// TIA Portal V19 export
FUNCTION "INTERLOCK DB" : Void   // FC17, LAD
{ S7_Optimized_Access := 'TRUE' }
// stored: SetENOAutomatically false
BEGIN

REGION Network 1: ERROR
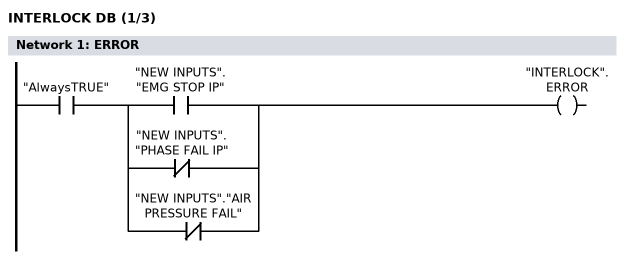
   RUNG wire#powerrail
      Contact( "AlwaysTRUE" )
      wire#w1
      Contact( "NEW INPUTS"."EMG STOP IP" )
      wire#w2
      Coil( "INTERLOCK".ERROR )
   END_RUNG
   RUNG wire#w1
      I_Contact( "NEW INPUTS"."PHASE FAIL IP" )
   END_RUNG wire#w2
   RUNG wire#w1
      I_Contact( "NEW INPUTS"."AIR PRESSURE FAIL" )
   END_RUNG wire#w2
   // the same network as SCL:
   "INTERLOCK".ERROR := "AlwaysTRUE" AND ("NEW INPUTS"."EMG STOP IP" OR NOT "NEW INPUTS"."PHASE FAIL IP" OR NOT "NEW INPUTS"."AIR PRESSURE FAIL");
END_REGION

REGION Network 2: MANUAL RESET
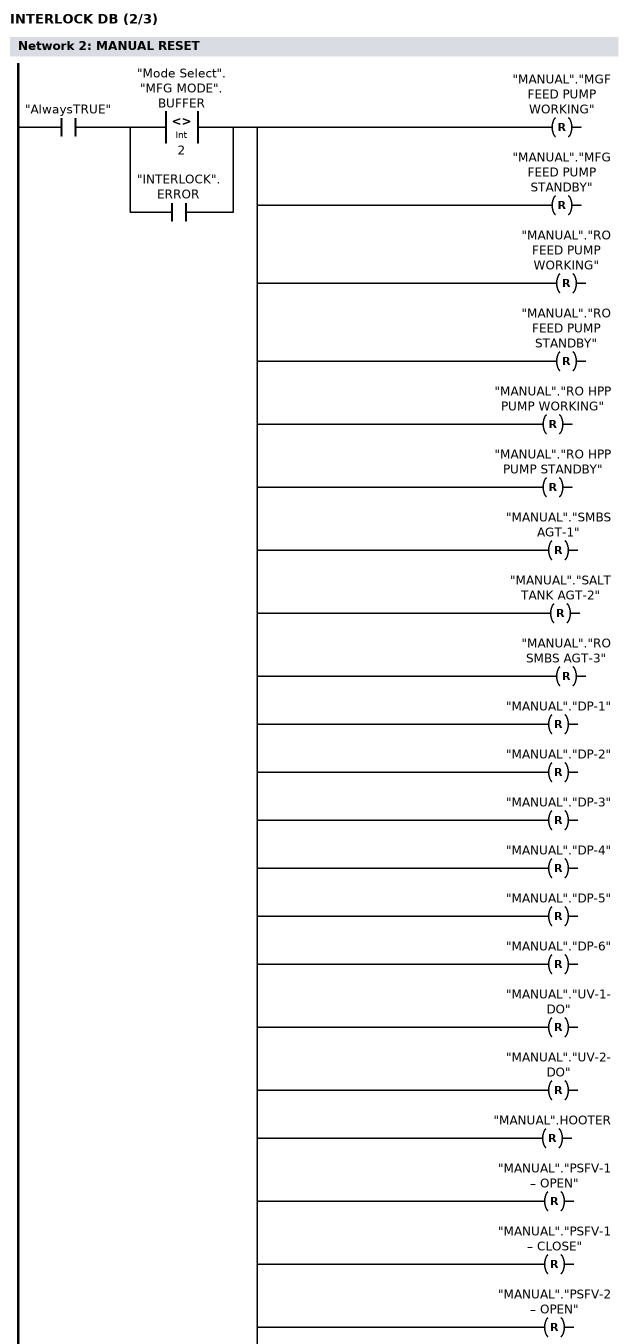
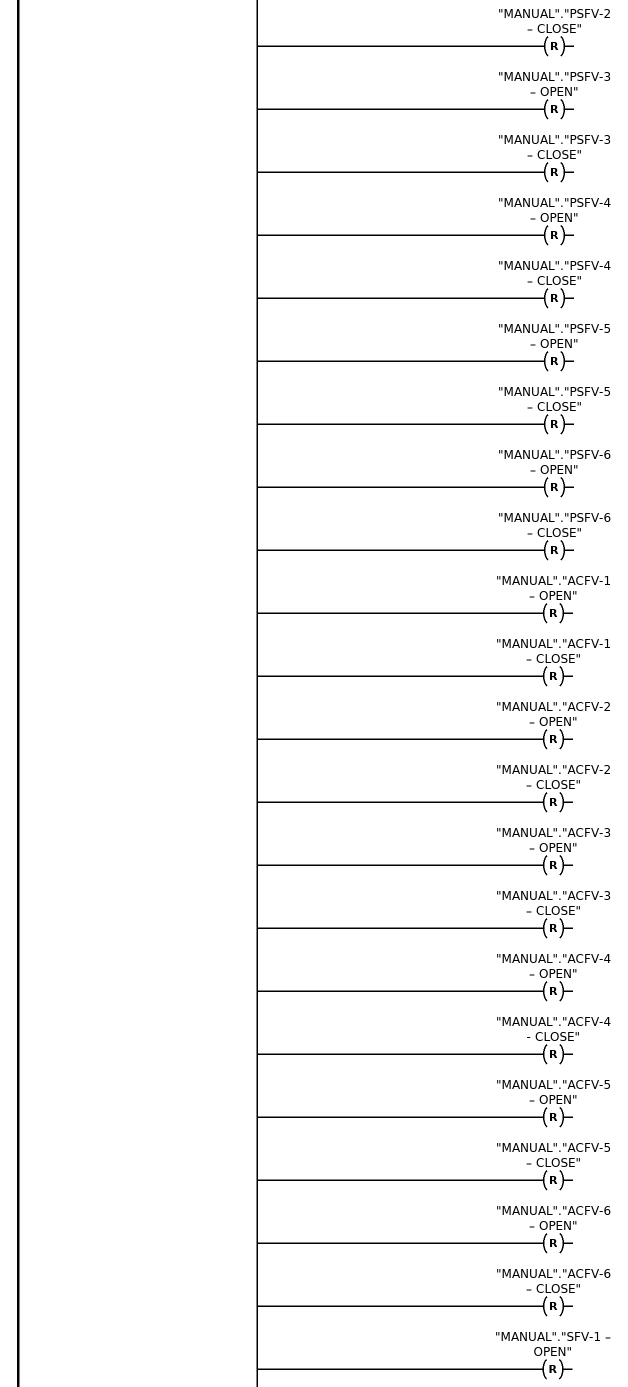
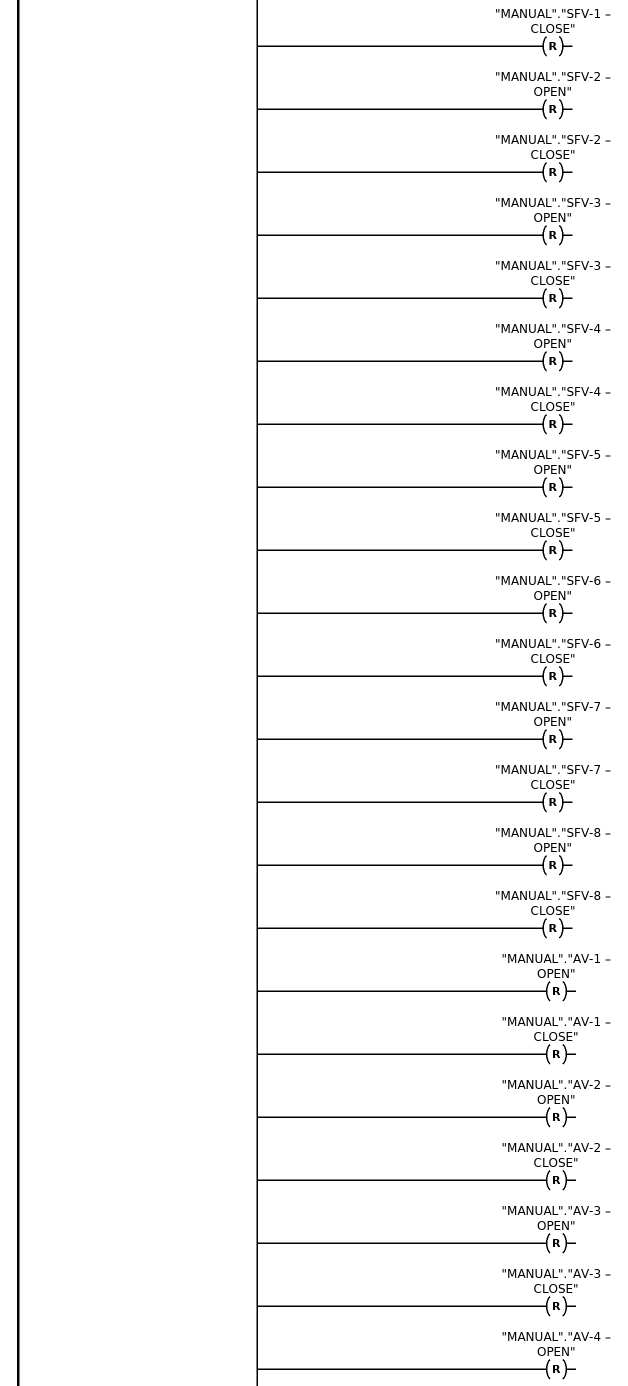
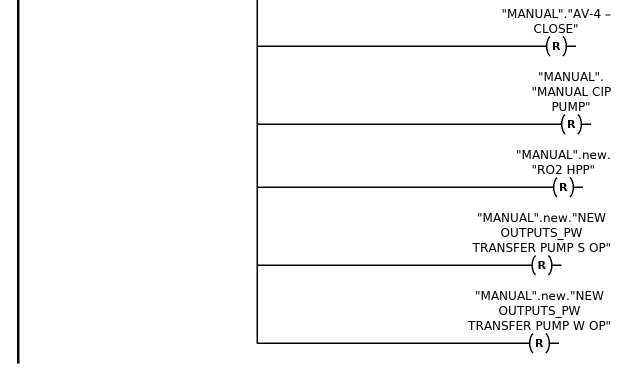
   RUNG wire#powerrail
      Contact( "AlwaysTRUE" )
      wire#w1
      { S7_Templates := "SrcType := Int" } NE_Contact(in1 := "Mode Select"."MFG MODE".BUFFER, in2 := 2)
      wire#w2
      R_Coil( "MANUAL"."MGF FEED PUMP WORKING" )
   END_RUNG
   RUNG wire#w1
      Contact( "INTERLOCK".ERROR )
   END_RUNG wire#w2
   RUNG wire#w2
      R_Coil( "MANUAL"."MFG FEED PUMP STANDBY" )
   END_RUNG
   RUNG wire#w2
      R_Coil( "MANUAL"."RO FEED PUMP WORKING" )
   END_RUNG
   RUNG wire#w2
      R_Coil( "MANUAL"."RO FEED PUMP STANDBY" )
   END_RUNG
   RUNG wire#w2
      R_Coil( "MANUAL"."RO HPP PUMP WORKING" )
   END_RUNG
   RUNG wire#w2
      R_Coil( "MANUAL"."RO HPP PUMP STANDBY" )
   END_RUNG
   RUNG wire#w2
      R_Coil( "MANUAL"."SMBS AGT-1" )
   END_RUNG
   RUNG wire#w2
      R_Coil( "MANUAL"."SALT TANK AGT-2" )
   END_RUNG
   RUNG wire#w2
      R_Coil( "MANUAL"."RO SMBS AGT-3" )
   END_RUNG
   RUNG wire#w2
      R_Coil( "MANUAL"."DP-1" )
   END_RUNG
   RUNG wire#w2
      R_Coil( "MANUAL"."DP-2" )
   END_RUNG
   RUNG wire#w2
      R_Coil( "MANUAL"."DP-3" )
   END_RUNG
   RUNG wire#w2
      R_Coil( "MANUAL"."DP-4" )
   END_RUNG
   RUNG wire#w2
      R_Coil( "MANUAL"."DP-5" )
   END_RUNG
   RUNG wire#w2
      R_Coil( "MANUAL"."DP-6" )
   END_RUNG
   RUNG wire#w2
      R_Coil( "MANUAL"."UV-1-DO" )
   END_RUNG
   RUNG wire#w2
      R_Coil( "MANUAL"."UV-2-DO" )
   END_RUNG
   RUNG wire#w2
      R_Coil( "MANUAL".HOOTER )
   END_RUNG
   RUNG wire#w2
      R_Coil( "MANUAL"."PSFV-1 – OPEN" )
   END_RUNG
   RUNG wire#w2
      R_Coil( "MANUAL"."PSFV-1 – CLOSE" )
   END_RUNG
   RUNG wire#w2
      R_Coil( "MANUAL"."PSFV-2 – OPEN" )
   END_RUNG
   RUNG wire#w2
      R_Coil( "MANUAL"."PSFV-2 – CLOSE" )
   END_RUNG
   RUNG wire#w2
      R_Coil( "MANUAL"."PSFV-3 – OPEN" )
   END_RUNG
   RUNG wire#w2
      R_Coil( "MANUAL"."PSFV-3 – CLOSE" )
   END_RUNG
   RUNG wire#w2
      R_Coil( "MANUAL"."PSFV-4 – OPEN" )
   END_RUNG
   RUNG wire#w2
      R_Coil( "MANUAL"."PSFV-4 – CLOSE" )
   END_RUNG
   RUNG wire#w2
      R_Coil( "MANUAL"."PSFV-5 – OPEN" )
   END_RUNG
   RUNG wire#w2
      R_Coil( "MANUAL"."PSFV-5 – CLOSE" )
   END_RUNG
   RUNG wire#w2
      R_Coil( "MANUAL"."PSFV-6 – OPEN" )
   END_RUNG
   RUNG wire#w2
      R_Coil( "MANUAL"."PSFV-6 – CLOSE" )
   END_RUNG
   RUNG wire#w2
      R_Coil( "MANUAL"."ACFV-1 – OPEN" )
   END_RUNG
   RUNG wire#w2
      R_Coil( "MANUAL"."ACFV-1 – CLOSE" )
   END_RUNG
   RUNG wire#w2
      R_Coil( "MANUAL"."ACFV-2 – OPEN" )
   END_RUNG
   RUNG wire#w2
      R_Coil( "MANUAL"."ACFV-2 – CLOSE" )
   END_RUNG
   RUNG wire#w2
      R_Coil( "MANUAL"."ACFV-3 – OPEN" )
   END_RUNG
   RUNG wire#w2
      R_Coil( "MANUAL"."ACFV-3 – CLOSE" )
   END_RUNG
   RUNG wire#w2
      R_Coil( "MANUAL"."ACFV-4 – OPEN" )
   END_RUNG
   RUNG wire#w2
      R_Coil( "MANUAL"."ACFV-4 - CLOSE" )
   END_RUNG
   RUNG wire#w2
      R_Coil( "MANUAL"."ACFV-5 – OPEN" )
   END_RUNG
   RUNG wire#w2
      R_Coil( "MANUAL"."ACFV-5 – CLOSE" )
   END_RUNG
   RUNG wire#w2
      R_Coil( "MANUAL"."ACFV-6 – OPEN" )
   END_RUNG
   RUNG wire#w2
      R_Coil( "MANUAL"."ACFV-6 – CLOSE" )
   END_RUNG
   RUNG wire#w2
      R_Coil( "MANUAL"."SFV-1 – OPEN" )
   END_RUNG
   RUNG wire#w2
      R_Coil( "MANUAL"."SFV-1 – CLOSE" )
   END_RUNG
   RUNG wire#w2
      R_Coil( "MANUAL"."SFV-2 – OPEN" )
   END_RUNG
   RUNG wire#w2
      R_Coil( "MANUAL"."SFV-2 – CLOSE" )
   END_RUNG
   RUNG wire#w2
      R_Coil( "MANUAL"."SFV-3 – OPEN" )
   END_RUNG
   RUNG wire#w2
      R_Coil( "MANUAL"."SFV-3 – CLOSE" )
   END_RUNG
   RUNG wire#w2
      R_Coil( "MANUAL"."SFV-4 – OPEN" )
   END_RUNG
   RUNG wire#w2
      R_Coil( "MANUAL"."SFV-4 – CLOSE" )
   END_RUNG
   RUNG wire#w2
      R_Coil( "MANUAL"."SFV-5 – OPEN" )
   END_RUNG
   RUNG wire#w2
      R_Coil( "MANUAL"."SFV-5 – CLOSE" )
   END_RUNG
   RUNG wire#w2
      R_Coil( "MANUAL"."SFV-6 – OPEN" )
   END_RUNG
   RUNG wire#w2
      R_Coil( "MANUAL"."SFV-6 – CLOSE" )
   END_RUNG
   RUNG wire#w2
      R_Coil( "MANUAL"."SFV-7 – OPEN" )
   END_RUNG
   RUNG wire#w2
      R_Coil( "MANUAL"."SFV-7 – CLOSE" )
   END_RUNG
   RUNG wire#w2
      R_Coil( "MANUAL"."SFV-8 – OPEN" )
   END_RUNG
   RUNG wire#w2
      R_Coil( "MANUAL"."SFV-8 – CLOSE" )
   END_RUNG
   RUNG wire#w2
      R_Coil( "MANUAL"."AV-1 – OPEN" )
   END_RUNG
   RUNG wire#w2
      R_Coil( "MANUAL"."AV-1 – CLOSE" )
   END_RUNG
   RUNG wire#w2
      R_Coil( "MANUAL"."AV-2 – OPEN" )
   END_RUNG
   RUNG wire#w2
      R_Coil( "MANUAL"."AV-2 – CLOSE" )
   END_RUNG
   RUNG wire#w2
      R_Coil( "MANUAL"."AV-3 – OPEN" )
   END_RUNG
   RUNG wire#w2
      R_Coil( "MANUAL"."AV-3 – CLOSE" )
   END_RUNG
   RUNG wire#w2
      R_Coil( "MANUAL"."AV-4 – OPEN" )
   END_RUNG
   RUNG wire#w2
      R_Coil( "MANUAL"."AV-4 – CLOSE" )
   END_RUNG
   RUNG wire#w2
      R_Coil( "MANUAL"."MANUAL CIP PUMP" )
   END_RUNG
   RUNG wire#w2
      R_Coil( "MANUAL".new."RO2 HPP" )
   END_RUNG
   RUNG wire#w2
      R_Coil( "MANUAL".new."NEW OUTPUTS_PW TRANSFER PUMP S OP" )
   END_RUNG
   RUNG wire#w2
      R_Coil( "MANUAL".new."NEW OUTPUTS_PW TRANSFER PUMP W OP" )
   END_RUNG
   // the same network as SCL:
   IF "AlwaysTRUE" AND (("Mode Select"."MFG MODE".BUFFER <> 2) OR "INTERLOCK".ERROR) THEN
       "MANUAL"."MGF FEED PUMP WORKING" := FALSE;
       "MANUAL"."MFG FEED PUMP STANDBY" := FALSE;
       "MANUAL"."RO FEED PUMP WORKING" := FALSE;
       "MANUAL"."RO FEED PUMP STANDBY" := FALSE;
       "MANUAL"."RO HPP PUMP WORKING" := FALSE;
       "MANUAL"."RO HPP PUMP STANDBY" := FALSE;
       "MANUAL"."SMBS AGT-1" := FALSE;
       "MANUAL"."SALT TANK AGT-2" := FALSE;
       "MANUAL"."RO SMBS AGT-3" := FALSE;
       "MANUAL"."DP-1" := FALSE;
       "MANUAL"."DP-2" := FALSE;
       "MANUAL"."DP-3" := FALSE;
       "MANUAL"."DP-4" := FALSE;
       "MANUAL"."DP-5" := FALSE;
       "MANUAL"."DP-6" := FALSE;
       "MANUAL"."UV-1-DO" := FALSE;
       "MANUAL"."UV-2-DO" := FALSE;
       "MANUAL".HOOTER := FALSE;
       "MANUAL"."PSFV-1 – OPEN" := FALSE;
       "MANUAL"."PSFV-1 – CLOSE" := FALSE;
       "MANUAL"."PSFV-2 – OPEN" := FALSE;
       "MANUAL"."PSFV-2 – CLOSE" := FALSE;
       "MANUAL"."PSFV-3 – OPEN" := FALSE;
       "MANUAL"."PSFV-3 – CLOSE" := FALSE;
       "MANUAL"."PSFV-4 – OPEN" := FALSE;
       "MANUAL"."PSFV-4 – CLOSE" := FALSE;
       "MANUAL"."PSFV-5 – OPEN" := FALSE;
       "MANUAL"."PSFV-5 – CLOSE" := FALSE;
       "MANUAL"."PSFV-6 – OPEN" := FALSE;
       "MANUAL"."PSFV-6 – CLOSE" := FALSE;
       "MANUAL"."ACFV-1 – OPEN" := FALSE;
       "MANUAL"."ACFV-1 – CLOSE" := FALSE;
       "MANUAL"."ACFV-2 – OPEN" := FALSE;
       "MANUAL"."ACFV-2 – CLOSE" := FALSE;
       "MANUAL"."ACFV-3 – OPEN" := FALSE;
       "MANUAL"."ACFV-3 – CLOSE" := FALSE;
       "MANUAL"."ACFV-4 – OPEN" := FALSE;
       "MANUAL"."ACFV-4 - CLOSE" := FALSE;
       "MANUAL"."ACFV-5 – OPEN" := FALSE;
       "MANUAL"."ACFV-5 – CLOSE" := FALSE;
       "MANUAL"."ACFV-6 – OPEN" := FALSE;
       "MANUAL"."ACFV-6 – CLOSE" := FALSE;
       "MANUAL"."SFV-1 – OPEN" := FALSE;
       "MANUAL"."SFV-1 – CLOSE" := FALSE;
       "MANUAL"."SFV-2 – OPEN" := FALSE;
       "MANUAL"."SFV-2 – CLOSE" := FALSE;
       "MANUAL"."SFV-3 – OPEN" := FALSE;
       "MANUAL"."SFV-3 – CLOSE" := FALSE;
       "MANUAL"."SFV-4 – OPEN" := FALSE;
       "MANUAL"."SFV-4 – CLOSE" := FALSE;
       "MANUAL"."SFV-5 – OPEN" := FALSE;
       "MANUAL"."SFV-5 – CLOSE" := FALSE;
       "MANUAL"."SFV-6 – OPEN" := FALSE;
       "MANUAL"."SFV-6 – CLOSE" := FALSE;
       "MANUAL"."SFV-7 – OPEN" := FALSE;
       "MANUAL"."SFV-7 – CLOSE" := FALSE;
       "MANUAL"."SFV-8 – OPEN" := FALSE;
       "MANUAL"."SFV-8 – CLOSE" := FALSE;
       "MANUAL"."AV-1 – OPEN" := FALSE;
       "MANUAL"."AV-1 – CLOSE" := FALSE;
       "MANUAL"."AV-2 – OPEN" := FALSE;
       "MANUAL"."AV-2 – CLOSE" := FALSE;
       "MANUAL"."AV-3 – OPEN" := FALSE;
       "MANUAL"."AV-3 – CLOSE" := FALSE;
       "MANUAL"."AV-4 – OPEN" := FALSE;
       "MANUAL"."AV-4 – CLOSE" := FALSE;
       "MANUAL"."MANUAL CIP PUMP" := FALSE;
       "MANUAL".new."RO2 HPP" := FALSE;
       "MANUAL".new."NEW OUTPUTS_PW TRANSFER PUMP S OP" := FALSE;
       "MANUAL".new."NEW OUTPUTS_PW TRANSFER PUMP W OP" := FALSE;
   END_IF;
END_REGION

REGION Network 3: TRANSFER PUMP WORKING & STANDBY
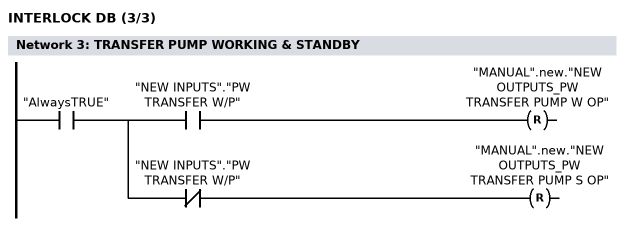
   RUNG wire#powerrail
      Contact( "AlwaysTRUE" )
      wire#w1
      Contact( "NEW INPUTS"."PW TRANSFER W/P" )
      R_Coil( "MANUAL".new."NEW OUTPUTS_PW TRANSFER PUMP W OP" )
   END_RUNG
   RUNG wire#w1
      I_Contact( "NEW INPUTS"."PW TRANSFER W/P" )
      R_Coil( "MANUAL".new."NEW OUTPUTS_PW TRANSFER PUMP S OP" )
   END_RUNG
   // the same network as SCL:
   IF "AlwaysTRUE" AND "NEW INPUTS"."PW TRANSFER W/P" THEN
       "MANUAL".new."NEW OUTPUTS_PW TRANSFER PUMP W OP" := FALSE;
   END_IF;
   IF "AlwaysTRUE" AND NOT "NEW INPUTS"."PW TRANSFER W/P" THEN
       "MANUAL".new."NEW OUTPUTS_PW TRANSFER PUMP S OP" := FALSE;
   END_IF;
END_REGION
END_FUNCTION
